FUNCTION_BLOCK ARRAY2VALUES_32_BYTE (* Service Interface Function Block Type *)
  (* Description: Copyright (c) 2014 Profactor GmbH, HR Agrartechnik GmbH This program and the accompanying materials are made available under the terms of the Eclipse Public License 2.0 which is available at https://www.eclipse.org/legal/epl-2.0/ SPDX-License-Identifier: EPL-2.0 *)
  (* Version 1.0, 2026-03-30, Franz Höpfinger, HR Agrartechnik GmbH, copy ARRAY2VALUES_2_LREAL and made this block *)
  PACKAGE eclipse4diac::convert;
  {SET_ATTRIBUTE(eclipse4diac::core::GenericClassName, 'GEN_ARRAY2VALUES')}
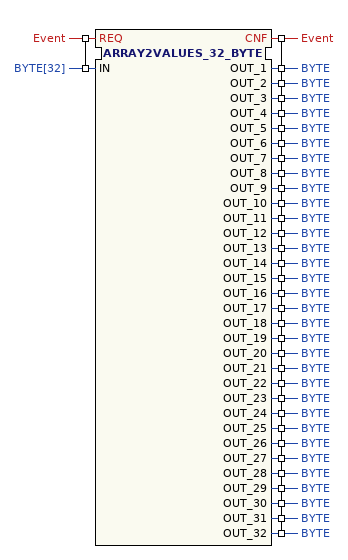
  EVENT_INPUT
    REQ WITH IN; (* Service Request *)
  END_EVENT
  EVENT_OUTPUT
    CNF WITH OUT_1, OUT_2, OUT_3, OUT_4, OUT_5, OUT_6, OUT_7, OUT_8, OUT_9, OUT_10, OUT_11, OUT_12, OUT_13, OUT_14, OUT_15, OUT_16, OUT_17, OUT_18, OUT_19, OUT_20, OUT_21, OUT_22, OUT_23, OUT_24, OUT_25, OUT_26, OUT_27, OUT_28, OUT_29, OUT_30, OUT_31, OUT_32; (* Confirmation of Requested Service *)
  END_EVENT
  VAR_INPUT
    IN : ARRAY [0..31] OF BYTE; (* Array input *)
  END_VAR
  VAR_OUTPUT
    OUT_1 : BYTE; (* output number 1 *)
    OUT_2 : BYTE; (* output number 2 *)
    OUT_3 : BYTE; (* output number 3 *)
    OUT_4 : BYTE; (* output number 4 *)
    OUT_5 : BYTE; (* output number 5 *)
    OUT_6 : BYTE; (* output number 6 *)
    OUT_7 : BYTE; (* output number 7 *)
    OUT_8 : BYTE; (* output number 8 *)
    OUT_9 : BYTE; (* output number 9 *)
    OUT_10 : BYTE; (* output number 10 *)
    OUT_11 : BYTE; (* output number 11 *)
    OUT_12 : BYTE; (* output number 12 *)
    OUT_13 : BYTE; (* output number 13 *)
    OUT_14 : BYTE; (* output number 14 *)
    OUT_15 : BYTE; (* output number 15 *)
    OUT_16 : BYTE; (* output number 16 *)
    OUT_17 : BYTE; (* output number 17 *)
    OUT_18 : BYTE; (* output number 18 *)
    OUT_19 : BYTE; (* output number 19 *)
    OUT_20 : BYTE; (* output number 20 *)
    OUT_21 : BYTE; (* output number 21 *)
    OUT_22 : BYTE; (* output number 22 *)
    OUT_23 : BYTE; (* output number 23 *)
    OUT_24 : BYTE; (* output number 24 *)
    OUT_25 : BYTE; (* output number 25 *)
    OUT_26 : BYTE; (* output number 26 *)
    OUT_27 : BYTE; (* output number 27 *)
    OUT_28 : BYTE; (* output number 28 *)
    OUT_29 : BYTE; (* output number 29 *)
    OUT_30 : BYTE; (* output number 30 *)
    OUT_31 : BYTE; (* output number 31 *)
    OUT_32 : BYTE; (* output number 32 *)
  END_VAR
END_FUNCTION_BLOCK
